PROGRAM MAIN
VAR
	Fan_Enable AT %Q* : BOOL;
END_VAR

END_PROGRAM

(* stored: Version 1.1.0.1, ProductVersion 3.1.4024.12
   POU MAIN: Id {5694769d-e5b0-4b4f-a601-0c181f66d836}, SpecialFunc None *)
